// TIA Portal V20 export
VAR_GLOBAL   // PLC tag table "Inputs Equipment"
   i_xSabload_Part1_p1_LR AT %I1.0 : Bool;   // Input - Sabload part 1 sensor - table P1 for Left and Right Jig
   i_xSabload_Part2_p1_L AT %I1.1 : Bool;   // Input - Sabload part 2 sensor - table P1 for Left Jig
   i_xSabload_Part3_p1_L AT %I1.2 : Bool;   // Input - Sabload part 3 sensor - table P1 for Left Jig
   i_xSabload_Part4_p1_LR AT %I1.3 : Bool;   // Input - Sabload part 4 sensor - table P1 for Left and Right Jig
   i_xSabload_Part2_p1_R AT %I1.4 : Bool;   // Input - Sabload part 2 sensor - table P1 for Right Jig
   i_xSabload_Part3_p1_R AT %I1.5 : Bool;   // Input - Sabload part 3 sensor - table P1 for Right Jig
   i_xSabload_Part1_p2_LR AT %I1.6 : Bool;   // Input - Sabload part 1 sensor - table P2 for Left and Right Jig
   i_xSabload_Part2_p2_L AT %I1.7 : Bool;   // Input - Sabload part 2 sensor - table P2 for Left Jig
   i_xSabload_Part3_p2_L AT %I2.0 : Bool;   // Input - Sabload part 3 sensor - table P2 for Left Jig
   i_xSabload_Part4_p2_LR AT %I2.1 : Bool;   // Input - Sabload part 4 sensor - table P2 for Left and Right Jig
   i_xSabload_Part2_p2_R AT %I2.2 : Bool;   // Input - Sabload part 2 sensor - table P2 for Right Jig
   i_xSabload_Part3_p2_R AT %I2.3 : Bool;   // Input - Sabload part 3 sensor - table P2 for Right Jig
   i_xBas342_ProgBit0 AT %I0.0 : Bool;   // Input - Bas 342 prog bit 0 for left side Jig
   i_xBas342_ProgBit1 AT %I0.1 : Bool;   // Input - Bas 342 prog bit 1 for Right side Jig
   i_xTableCheck_JigPresent_p1 AT %I0.2 : Bool;   // Input: TableCheck process 1 Sensor for Jig presence for Table P1
   i_xTableCheck_JigPresent_p2 AT %I0.3 : Bool;   // Input: TableCheck process 1 Sensor for Jig presence for Table P2
END_VAR
